	DATA_BLOCK DB2053
	TITLE =Event DB : LINE 1 SEC 23 GERM 7
	//
	//COPYRIGHT:    (C) 2006 BY  BUHLER AG
	//                           CH-9240 UZWIL  SWITZERLAND
	//
	//PRODUCT:      WinCoS_BIW01_09
	//
	//TITLE:        Event DB : LINE 1 SEC 23 GERM 7
	//
	//
	//
	//
	//-------------------------------------------------------------------------
	//
	//IDENT:        AUTHOR:             DEPT:                       DATE:
	//
	//P01_DB000.1.0 K.Renz              CSB41                       21.Okt.2009
	//              1st Release
	//
	//--------------------------------------------------------------------------------
	//
	//PURPOSE: SIS Line specific parameters and values
	//
	//MANUAL :
	//
	//CODE   :
	//
	//RESTRICTIONS:
	//
	//--------------------------------------------------------------------------------
	//
	//
	//
	AUTHOR  : KR
	FAMILY  : ASW

	VERSION : 0.0
	"SSA_MH_EventsToPIC"
	BEGIN
	END_DATA_BLOCK
